FUNCTION SCALE_LIM (* Scaling Function Block with limits *)
  (* Standard: 61499-1; Description: Copyright (c) 2024 HR Agrartechnik GmbH This program and the accompanying materials are made available under the terms of the Eclipse Public License 2.0 which is available at https://www.eclipse.org/legal/epl-2.0/ SPDX-License-Identifier: EPL-2.0 *)
  (* Version 1.0, 2024-09-19, Franz Höpfinger, HR Agrartechnik GmbH *)
  (* Version 3.0, 2025-04-14, Patrick Aigner, changed package *)
  PACKAGE eclipse4diac::signalprocessing;
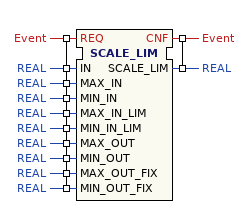
  EVENT_INPUT
    REQ WITH IN, MAX_IN, MIN_IN, MAX_IN_LIM, MIN_IN_LIM, MAX_OUT, MIN_OUT, MAX_OUT_FIX, MIN_OUT_FIX;
  END_EVENT
  EVENT_OUTPUT
    CNF WITH SCALE_LIM;
  END_EVENT
  VAR_INPUT
    IN : REAL; (* Input to be Scaled *)
    MAX_IN : REAL; (* Maximum Input *)
    MIN_IN : REAL; (* Minimum Input *)
    MAX_IN_LIM : REAL; (* Maximum Input Limit, if IN is bigger, Output is MAX2_ESC *)
    MIN_IN_LIM : REAL; (* Minimum Input Limit, if IN is smaller, Output is MIN2_ESC *)
    MAX_OUT : REAL; (* Maximum Ouput *)
    MIN_OUT : REAL; (* Minimum Output *)
    MAX_OUT_FIX : REAL; (* Maximum Ouput Fix Value, ist set if IN is bigger than MAX_IN_LIM *)
    MIN_OUT_FIX : REAL; (* Minimum Output Fix Value, ist set if IN is smaller than MIN_IN_LIM *)
  END_VAR
  VAR_OUTPUT
    SCALE_LIM : REAL;
  END_VAR
  BODY IN ST:
PACKAGE signalprocessing;

(* Scaling Function Block with limits *)
FUNCTION SCALE_LIM : REAL
VAR_INPUT
	IN : REAL;    // Input to be Scaled
	MAX_IN : REAL;    // Maximum Input
	MIN_IN : REAL;    // Minimum Input
	MAX_IN_LIM : REAL;    // Maximum Input Limit, if IN is bigger, Output is MAX2_ESC
	MIN_IN_LIM : REAL;    // Minimum Input Limit, if IN is smaller, Output is MIN2_ESC
	MAX_OUT : REAL;    // Maximum Ouput
	MIN_OUT : REAL;    // Minimum Output
	MAX_OUT_FIX : REAL;    // Maximum Ouput Fix Value, ist set if IN is bigger than MAX_IN_LIM
	MIN_OUT_FIX : REAL;    // Minimum Output Fix Value, ist set if IN is smaller than MIN_IN_LIM
END_VAR

IF (IN < MIN_IN_LIM) THEN
	SCALE_LIM := MIN_OUT_FIX;
ELSIF (IN> MAX_IN_LIM) THEN
	SCALE_LIM := MAX_OUT_FIX;
ELSE
	SCALE_LIM := (IN - MIN_IN) * (MAX_OUT - MIN_OUT) / (MAX_IN - MIN_IN) + MIN_OUT;
END_IF;

END_FUNCTION
  END_BODY
END_FUNCTION
